// TIA Portal V17 export
// export: Created 2024-09-15T12:30:11.7290918Z, ExportSetting WithDefaults, DisplayName Totally Integrated Automation Portal, DisplayVersion V17, DisplayName TIA Portal Openness, DisplayVersion V17, DisplayName TIA Portal Version Control Interface, DisplayVersion V17, DisplayName STEP 7 Professional, DisplayVersion V17, DisplayName STEP 7 Safety, DisplayVersion V17, DisplayName WinCC Professional, DisplayVersion V17
DATA_BLOCK "DPS_Tracking_DB"   // DB51
VERSION : 0.1
// stored: AutoNumber true, DBAccessibleFromOPCUA true, DBAccessibleFromWebserver true, InstanceOfName DPS_Tracking, InstanceOfType FB
"DPS_Tracking"
   // VAR
   //    Location : String;
   // END_VAR
BEGIN
END_DATA_BLOCK
